# EPICS substitutions: ecmcApp/Db/SlitX-xp.substitutions
file "ecmc.template" {
pattern
{P,        N,  M,   R,     DTYP,         PORT,     ADDR,  DESC,          EGU, DIR,  VELO, HVEL, JVEL,  JAR,  VBAS,  ACCL,  BDST, DLY,  BVEL,  BACC,  MRES,      ERES,       PREC,  DLLM,  DHLM,  INIT}
{"IOC2:",  1,  xp,  xp-,  "asynMotor",   MCU1,     1,     "XPosition",   mm,  Pos,  10,   5,    10,    10.2, 0,     1,     0,    0.3,  1,     .2,    0.0046875  0.01754386  3,     0,     0,     ""}
}
